// TIA Portal V16 export
// export: Created 2021-04-11T09:51:28.6139801Z, ExportSetting WithDefaults, DisplayName Totally Integrated Automation Portal, DisplayVersion V16, DisplayName TIA Portal Version Control Interface, DisplayVersion V16, DisplayName TIA Portal Openness, DisplayVersion V16, DisplayName STEP 7 Professional, DisplayVersion V16, DisplayName STEP 7 Safety, DisplayVersion V16, DisplayName WinCC Unified SCADA Engineering System, DisplayVersion V16
DATA_BLOCK "ManualMode_DB"   // DB30
VERSION : 0.1
// stored: AutoNumber false, DBAccessibleFromOPCUA true, InstanceOfName ManualMode, InstanceOfType FB
"ManualMode"
   // VAR
   //    Bunker_Left : Array[0..12] of "controlValve";
   //    Bunker_Right : Array[0..12] of "controlValve";
   //    Door : Array[0..12] of "controlValve";
   //    flipper : "controlValve";
   //    runAll : Struct
   //       vibroLot : Bool;
   //    END_STRUCT;
   //    stopAlarm : Bool;
   // END_VAR
BEGIN
END_DATA_BLOCK
